TYPE ST_DigitalOut :
STRUCT
	dout 		: BOOL;
	dout_fdbk			: BOOL;
END_STRUCT
END_TYPE

(* stored: Version 1.1.0.1, ProductVersion 3.1.4024.12
   DUT ST_DigitalOut: Id {7e3a32d5-f433-446a-9a84-2322628ec4d7} *)
